FUNCTION_BLOCK _DWORD_TestSuite EXTENDS TcUnit.FB_TestSuite
VAR
END_VAR

TestAddress();
TestClearReference();
TestClone();
TestTypeNameReturnsExpected();
TestIsFloat();
TestIsSigned();
TestMakeReferenceToFollowsReference();
TestMakeReferenceToUpdatesReference();
TestSize();
TestValueReturnsExpectedAfterInit();
TestValueReturnsExpectedAfterChange();
TestSerializeTypeWith();
TestSerializeWith();
TestTryDeserializeFrom();
TestTryMakeReferenceToFollowsReference();
TestTryMakeReferenceToUpdatesReference();

METHOD PUBLIC TestAddress
VAR
    _type : _DWORD(0);
    notExpected : PVOID := 0;
    actual : PVOID;
END_VAR
TEST('TestAddress');

actual := _type.Address;

AssertFalse(
    Condition := (notExpected = actual),
    Message := 'Type did not return a valid address.'
);

TEST_FINISHED();
END_METHOD

METHOD PUBLIC TestClearReference
VAR
    _type : _DWORD(0);
	target : DWORD := 0;
    expected : DWORD := 0;
    actual : DWORD;
END_VAR
TEST('TestClearReference');

_type.MakeReferenceTo(target);
_type.ClearReference();
target := 123;

actual := _type.Value;

AssertEquals(
    Expected := expected,
    Actual := actual,
    Message := 'Value did not follow target change'
);

TEST_FINISHED();
END_METHOD

METHOD PUBLIC TestClone
VAR
    _type : _DWORD(123);
	clone : I_Datatype;
	isValidClone : BOOL;
	compareResult : DINT;
END_VAR
TEST('TestClone');

clone := _type.Clone();

isValidClone := clone <> 0;

IF isValidClone THEN
	compareResult := memcmp(_type.Address, clone.Address, clone.Size);
END_IF

AssertTrue(
	Condition := isValidClone,
	Message := 'Clone did not produce a clone'
);

AssertEquals_DINT(
	Expected := 0,
    Actual := compareResult,
    Message := 'Clone did not return a valid clone.'
);

clone.Dispose();

TEST_FINISHED();
END_METHOD

METHOD PUBLIC TestIsFloat
VAR
    _type : _DWORD(0);
END_VAR
TEST('TestIsFloat');

AssertFalse(
	Condition := _type.IsFloat,
    Message := 'Type did not correctly identify itself as being unsigned'
);

TEST_FINISHED();
END_METHOD

METHOD PUBLIC TestIsSigned
VAR
    _type : _DWORD(0);
END_VAR
TEST('TestIsSigned');

AssertFalse(
	Condition := _type.IsSigned,
    Message := 'Type did not correctly identify itself as being unsigned'
);

TEST_FINISHED();
END_METHOD

METHOD PUBLIC TestMakeReferenceToFollowsReference
VAR
    _type : _DWORD(0);
	target : DWORD := 0;
    expected : DWORD := 123;
    actual : DWORD;
END_VAR
TEST('TestMakeReferenceToFollowsReference');

_type.MakeReferenceTo(target);
target := 123;

actual := _type.Value;

AssertEquals(
    Expected := expected,
    Actual := actual,
    Message := 'Value did not follow target change'
);

TEST_FINISHED();
END_METHOD

METHOD PUBLIC TestMakeReferenceToUpdatesReference
VAR
    _type : _DWORD(0);
	target : DWORD := 0;
    expected : DWORD := 123;
    actual : DWORD;
END_VAR
TEST('TestMakeReferenceToUpdatesReference');

_type.MakeReferenceTo(target);
_type.Value := 123;

actual := target;

AssertEquals(
    Expected := expected,
    Actual := actual,
    Message := 'Value did not update target'
);

TEST_FINISHED();
END_METHOD

METHOD PUBLIC TestSerializeTypeWith
VAR
    _type : _DWORD(0);
    serializer : JsonSerializer;
    expected : STRING(500) := '{"typeName":"DWORD","minValue":0,"maxValue":4294967295,"isSigned":false,"isFloat":false}';
    actual : STRING(500);
END_VAR
TEST('TestSerializeTypeWith');

serializer.Reset();
_type.SerializeTypeWith(serializer);
serializer.TryGetSerializedData(ADR(actual), SIZEOF(actual));

AssertEquals_STRING(
    Expected := expected,
    Actual := actual,
    Message := 'Serialization of type did not return correct string.'
);

TEST_FINISHED();
END_METHOD

METHOD PUBLIC TestSerializeWith
VAR
    _type : _DWORD(65535);
    serializer : JsonSerializer;
    expected : STRING := '65535';
    actual : STRING(500);
END_VAR
TEST('TestSerializeWith');

serializer.Reset();
_type.SerializeWith(serializer);
serializer.TryGetSerializedData(ADR(actual), SIZEOF(actual));

AssertEquals_STRING(
    Expected := expected,
    Actual := actual,
    Message := 'Serialization of type data did not return correct string.'
);

TEST_FINISHED();
END_METHOD

METHOD PUBLIC TestSize
VAR
    _type : _DWORD(0);
    expected : UDINT := SIZEOF(DWORD);
    actual : UDINT;
END_VAR
TEST('TestSize');

actual := _type.Size;

AssertEquals_UDINT(
    Expected := Expected,
    Actual := actual,
    Message := 'Type did not return the correct size.'
);

TEST_FINISHED();
END_METHOD

METHOD PUBLIC TestTryDeserializeFrom
VAR
    deserializer : JsonDeserializer;
    feedback : DeserializerFeedback;
    json : STRING := '65535';
    _type : _DWORD(0);
    expected : DWORD := 65535;
    actual : DWORD;
 END_VAR
TEST('TestTryDeserializeFrom');

deserializer.Reset();
deserializer.TryLoad(json);
_type.TryDeserializeFrom(Deserializer, Feedback);

actual := _type.Value;

AssertEquals(
    Expected := expected,
    Actual := actual,
    Message := 'Type did not deserialize correctly.'
);

TEST_FINISHED();
END_METHOD

METHOD PUBLIC TestTryMakeReferenceToFollowsReference
VAR
    _type : _DWORD(0);
	target : _DWORD(0);
    expected : DWORD := 123;
    actual : DWORD;
END_VAR
TEST('TestTryMakeReferenceToFollowsReference');

_type.TryMakeReferenceTo(target);
target.Value := 123;

actual := _type.Value;

AssertEquals(
    Expected := expected,
    Actual := actual,
    Message := 'Value did not follow target change'
);

TEST_FINISHED();
END_METHOD

METHOD PUBLIC TestTryMakeReferenceToUpdatesReference
VAR
    _type : _DWORD(0);
	target : _DWORD(0);
    expected : DWORD := 123;
    actual : DWORD;
END_VAR
TEST('TestTryMakeReferenceToUpdatesReference');

_type.TryMakeReferenceTo(target);
_type.Value := 123;

actual := target.Value;

AssertEquals(
    Expected := expected,
    Actual := actual,
    Message := 'Value did not update target'
);

TEST_FINISHED();
END_METHOD

METHOD PUBLIC TestTypeNameReturnsExpected
VAR
    _type : _DWORD(0);
    expected : STRING := 'DWORD';
    actual : STRING;
END_VAR
TEST('TestTypeNameReturnsExpected');

actual := _type.TypeName;

AssertEquals_STRING(
    Expected := expected,
    Actual := actual,
    Message := 'Type did not return correct iec type.'
);

TEST_FINISHED();
END_METHOD

METHOD PUBLIC TestValueReturnsExpectedAfterChange
VAR
    _type : _DWORD(0);
    expected : DWORD := 65535;
    actual : DWORD;
END_VAR
TEST('TestValueReturnsExpectedAfterChange');

_type.Value := 65535;

actual := _type.Value;

AssertEquals(
    Expected := expected,
    Actual := actual,
    Message := 'Expected value not returned after change.'
);

TEST_FINISHED();
END_METHOD

METHOD PUBLIC TestValueReturnsExpectedAfterInit
VAR
    _type : _DWORD(65535);
    expected : DWORD := 65535;
    actual : DWORD;
END_VAR
TEST('TestValueReturnsExpectedAfterInit');

actual := _type.Value;

AssertEquals(
    Expected := expected,
    Actual := actual,
    Message := 'Expected value not returned after Init.'
);

TEST_FINISHED();
END_METHOD

END_FUNCTION_BLOCK

(* stored: Version 1.1.0.1, ProductVersion 3.1.4024.12
   POU _DWORD_TestSuite: Id {0699e8b0-837e-4c73-b147-696e2a911cbe}, SpecialFunc None
   Method TestAddress: Id {84aef0fa-be01-493a-b53f-1c3d2c37df1c}
   Method TestClearReference: Id {d9760088-2d9e-44ba-9aff-7f3ea3028722}
   Method TestClone: Id {8d5824d5-4dca-4a5a-a6e9-7bc01a358612}
   Method TestIsFloat: Id {7d0d291c-7943-0378-3b93-4f3a318657c2}
   Method TestIsSigned: Id {34cc1a80-5ee5-4fbe-86fd-8833af375397}
   Method TestMakeReferenceToFollowsReference: Id {f9810f6c-70f4-4a29-b381-c4697eeeffb3}
   Method TestMakeReferenceToUpdatesReference: Id {56e6b56f-c696-46f9-95c1-1afcf6a73e5b}
   Method TestSerializeTypeWith: Id {939d934f-cebf-41b8-a7e9-3145dd034c91}
   Method TestSerializeWith: Id {482c3cd0-82b5-4e2b-a610-f77ccfff1220}
   Method TestSize: Id {c3db0f6e-7a61-4152-96b1-af5bddd025f1}
   Method TestTryDeserializeFrom: Id {f8f6af42-c776-4405-a4e4-f5248d65513e}
   Method TestTryMakeReferenceToFollowsReference: Id {dfb5c83f-800a-478b-82a8-5d63fd633acc}
   Method TestTryMakeReferenceToUpdatesReference: Id {5147fb98-ef62-40f1-8447-a25cb6d0ca25}
   Method TestTypeNameReturnsExpected: Id {727f6dd7-ad0e-420d-8bb5-ad9767f1e26a}
   Method TestValueReturnsExpectedAfterChange: Id {868ef3f5-fc17-4417-82fd-0b7adf2caf74}
   Method TestValueReturnsExpectedAfterInit: Id {38d0a794-504a-4a31-b35c-1fc3533be003} *)
